// TIA Portal V17 export
// export: Created 2022-07-20T06:59:39.1268711Z, ExportSetting WithDefaults, DisplayName Totally Integrated Automation Portal, DisplayVersion V17, DisplayName TIA Portal Openness, DisplayVersion V17, DisplayName TIA Portal Version Control Interface, DisplayVersion V17, DisplayName SINAMICS Startdrive Advanced, DisplayVersion V17, DisplayName SINAMICS Startdrive G130, G150, S120, S150, SINAMICS MV, S210, DisplayVersion V17, DisplayName SINAMICS Startdrive G110M, G120, G120C, G120D, G120P, G115D, DisplayVersion V17, DisplayName STEP 7 Professional, DisplayVersion V17, DisplayName STEP 7 Safety, DisplayVersion V17, DisplayName WinCC Advanced, DisplayVersion V17
FUNCTION "FC10012_2IntToDint" : Void   // FC10012, LAD
TITLE = FC10012_2IntToDint
{ S7_Optimized_Access := 'TRUE' }
AUTHOR : Anirouddh
FAMILY : 1001x_CONVERT
VERSION : 1.0
// Release note : 
// 1.0 - Feature developped
// stored: AutoNumber false, IsIECCheckEnabled false, SetENOAutomatically false, UDAEnableTagReadback false
   VAR_INPUT
      HighInt : Int;
      LowInt : Int;
   END_VAR
   VAR_OUTPUT
      Output_DInt : DInt;
   END_VAR
   VAR_TEMP
      Temp1 : DWord;
      Temp2 : DWord;
   END_VAR
BEGIN

REGION Network 1 (SCL): 2 Ints To Dint Conversion
   #Temp1 := INT_TO_DWORD(#HighInt);
   #Temp2 := INT_TO_DWORD(#LowInt);

   #Temp1 := SHL_DWORD(IN := #Temp1, N := 16);

   #Temp1 := #Temp1 OR #Temp2;

   #Output_DInt := DWORD_TO_DINT(#Temp1);
END_REGION
END_FUNCTION
